DATA_BLOCK "HMIInterchange"
{ S7_Optimized_Access := 'TRUE' }
VERSION : 0.1
NON_RETAIN
   VAR
      operation : Struct
         add : Bool;
         subtract : Bool;
         multiply : Bool;
         divide : Bool;
      END_STRUCT;
      values : Struct
         value1 : Int;
         value2 : Int;
         result : Int;
      END_STRUCT;
      "counter" : Struct
         reset : Bool;
         counterValue : Int;
      END_STRUCT;
      shutdown : Struct
         start : Bool;
         returnValue : Word;
      END_STRUCT;
   END_VAR


BEGIN

END_DATA_BLOCK

